// Mitsubishi GX Works2 project: 20240228_AI机RTU测试   PLC: FX3S

PROGRAM MAIN
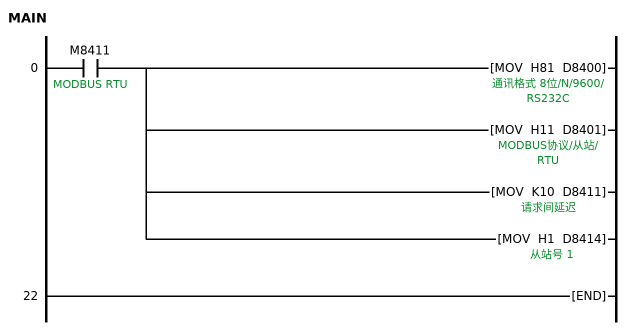
0     LD      M8411  ; MODBUS RTU
      MOV     H81 D8400  ; 通讯格式 8位/N/9600/RS232C
      MOV     H11 D8401  ; MODBUS协议/从站/RTU
      MOV     K10 D8411  ; 请求间延迟
      MOV     H1 D8414  ; 从站号 1
22    END
END_PROGRAM

// device comments not shown above
X001  ; 运行准备X1
X002  ; 启动按键X2
X003  ; 复位按键X3
X005  ; 小径对焦
X006  ; 大径对焦-旋钮
X007  ; 小径对焦-旋钮
X010  ; DAM-OUT1-NO
X011  ; DAM-OUT2-NO
X012  ; DAM-OUT3-NO
X013  ; DAM-OUT4-NO
X014  ; DAM-OUT5-NO
X015  ; DAM-OUT6-NO
M0  ; 运行准备
M1  ; 启动运转
M2  ; 伺服ON
M3  ; 复位
M6  ; 大径对焦
M7  ; 小径对焦
Y000  ; 伺服输出
Y001  ; 准备LED
Y002  ; 启动LED
Y003  ; 复位LED
Y004  ; 气缸后退
Y005  ; 气缸前进
Y006  ; 气缸前进
Y007  ; 气缸后退
Y012  ; 黄色LED
Y013  ; 绿色LED
Y014  ; 红色LED
Y015  ; 运行中
